Staubli VAL3: onSave.pgx

public program onSave()
begin
  sml:libSave()
  big:libSave()
end
